FUNCTION_BLOCK FB_MixingVR01
VAR_INPUT
	bEnable 	: BOOL; //uruchom mieszanie z zadaną czestotliwościa pracy
	rSpeedAuto	: REAL; //zadana częstotliwość pracy M01 i M02	
END_VAR
VAR_OUTPUT
	bCmd_M01	: BOOL;
	bCmd_M02    : BOOL;
	rSpeedSet	: REAL;
END_VAR

// ---------------------------------------------------------
// STOP GLOBALNY
// ---------------------------------------------------------
IF NOT bEnable THEN
	rSpeedAuto := 0.0;
	bCmd_M01 := FALSE;
	bCmd_M02 := FALSE;
ELSE
	rSpeedSet := rSpeedAuto;
	bCmd_M01 := TRUE;
	bCmd_M02 := TRUE;
END_IF

END_FUNCTION_BLOCK

(* stored: Version 1.1.0.1, ProductVersion 3.1.4024.16
   POU FB_MixingVR01: Id {a23967ff-349c-49ab-ba77-9ea5a940b929}, SpecialFunc None *)
